// Mitsubishi GX Works2 project: NIAP1546_0600_IC-1M_R2   PLC: FX3S

PROGRAM MAIN
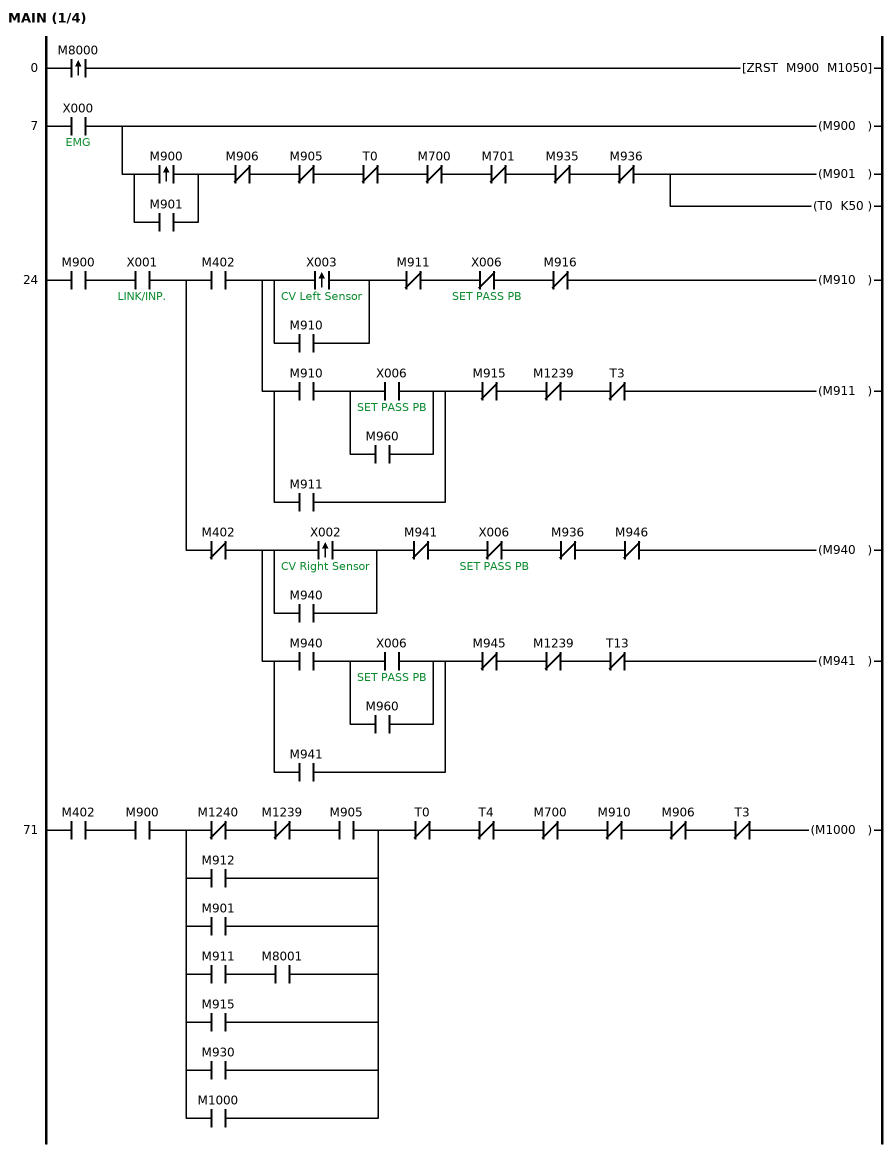
0     LDP     M8000
      ZRST    M900 M1050
7     LD      X000  ; EMG
      OUT     M900
      LDP     M900
      OR      M901
      ANB
      ANI     M906
      ANI     M905
      ANI     T0
      ANI     M700
      ANI     M701
      ANI     M935
      ANI     M936
      OUT     M901
      OUT     T0 K50
24    LD      M900
      AND     X001  ; LINK/INP.
      MPS
      AND     M402
      MPS
      LDP     X003  ; CV Left Sensor
      OR      M910
      ANB
      ANI     M911
      ANI     X006  ; SET PASS PB
      ANI     M916
      OUT     M910
      MPP
      LD      M910
      LD      X006  ; SET PASS PB
      OR      M960
      ANB
      OR      M911
      ANB
      ANI     M915
      ANI     M1239
      ANI     T3
      OUT     M911
      MPP
      ANI     M402
      MPS
      LDP     X002  ; CV Right Sensor
      OR      M940
      ANB
      ANI     M941
      ANI     X006  ; SET PASS PB
      ANI     M936
      ANI     M946
      OUT     M940
      MPP
      LD      M940
      LD      X006  ; SET PASS PB
      OR      M960
      ANB
      OR      M941
      ANB
      ANI     M945
      ANI     M1239
      ANI     T13
      OUT     M941
71    LD      M402
      AND     M900
      LDI     M1240
      ANI     M1239
      AND     M905
      OR      M912
      OR      M901
      LD      M911
      AND     M8001
      ORB
      OR      M915
      OR      M930
      OR      M1000
      ANB
      ANI     T0
      ANI     T4
      ANI     M700
      ANI     M910
      ANI     M906
      ANI     T3
      OUT     M1000
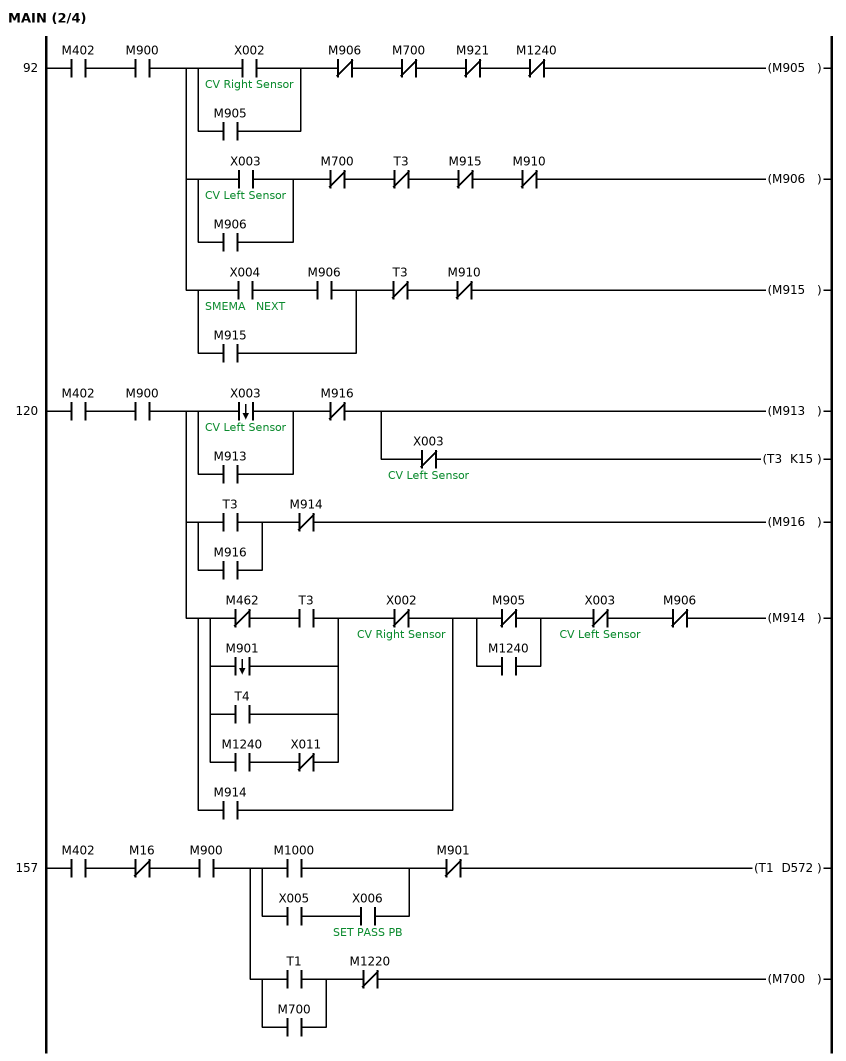
92    LD      M402
      AND     M900
      MPS
      LD      X002  ; CV Right Sensor
      OR      M905
      ANB
      ANI     M906
      ANI     M700
      ANI     M921
      ANI     M1240
      OUT     M905
      MRD
      LD      X003  ; CV Left Sensor
      OR      M906
      ANB
      ANI     M700
      ANI     T3
      ANI     M915
      ANI     M910
      OUT     M906
      MPP
      LD      X004  ; SMEMA   NEXT
      AND     M906
      OR      M915
      ANB
      ANI     T3
      ANI     M910
      OUT     M915
120   LD      M402
      AND     M900
      MPS
      LDF     X003  ; CV Left Sensor
      OR      M913
      ANB
      ANI     M916
      OUT     M913
      ANI     X003  ; CV Left Sensor
      OUT     T3 K15
      MRD
      LD      T3
      OR      M916
      ANB
      ANI     M914
      OUT     M916
      MPP
      LDI     M462
      AND     T3
      ORF     M901
      OR      T4
      LD      M1240
      ANI     X011
      ORB
      ANI     X002  ; CV Right Sensor
      OR      M914
      ANB
      LDI     M905
      OR      M1240
      ANB
      ANI     X003  ; CV Left Sensor
      ANI     M906
      OUT     M914
157   LD      M402
      ANI     M16
      AND     M900
      MPS
      LD      M1000
      LD      X005
      AND     X006  ; SET PASS PB
      ORB
      ANB
      ANI     M901
      OUT     T1 D572
      MPP
      LD      T1
      OR      M700
      ANB
      ANI     M1220
      OUT     M700
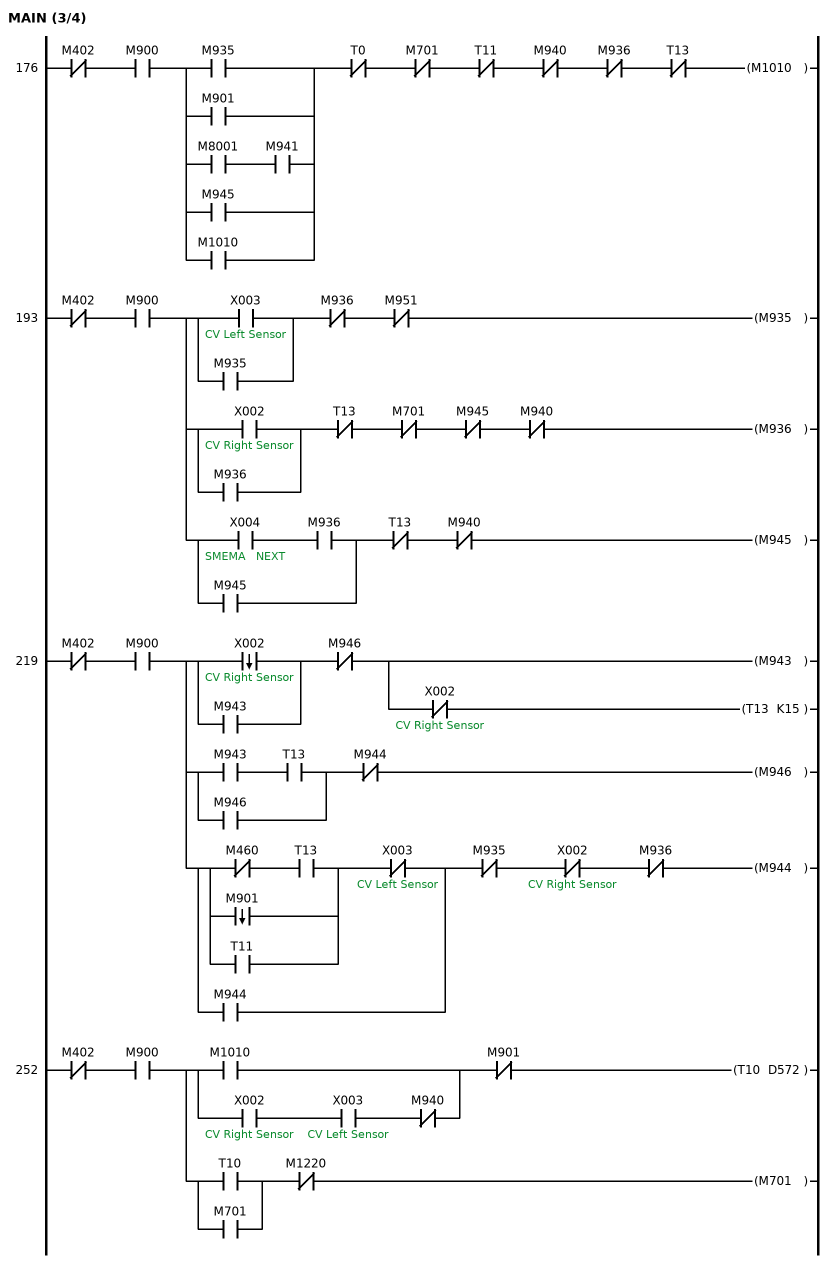
176   LDI     M402
      AND     M900
      LD      M935
      OR      M901
      LD      M8001
      AND     M941
      ORB
      OR      M945
      OR      M1010
      ANB
      ANI     T0
      ANI     M701
      ANI     T11
      ANI     M940
      ANI     M936
      ANI     T13
      OUT     M1010
193   LDI     M402
      AND     M900
      MPS
      LD      X003  ; CV Left Sensor
      OR      M935
      ANB
      ANI     M936
      ANI     M951
      OUT     M935
      MRD
      LD      X002  ; CV Right Sensor
      OR      M936
      ANB
      ANI     T13
      ANI     M701
      ANI     M945
      ANI     M940
      OUT     M936
      MPP
      LD      X004  ; SMEMA   NEXT
      AND     M936
      OR      M945
      ANB
      ANI     T13
      ANI     M940
      OUT     M945
219   LDI     M402
      AND     M900
      MPS
      LDF     X002  ; CV Right Sensor
      OR      M943
      ANB
      ANI     M946
      OUT     M943
      ANI     X002  ; CV Right Sensor
      OUT     T13 K15
      MRD
      LD      M943
      AND     T13
      OR      M946
      ANB
      ANI     M944
      OUT     M946
      MPP
      LDI     M460
      AND     T13
      ORF     M901
      OR      T11
      ANI     X003  ; CV Left Sensor
      OR      M944
      ANB
      ANI     M935
      ANI     X002  ; CV Right Sensor
      ANI     M936
      OUT     M944
252   LDI     M402
      AND     M900
      MPS
      LD      M1010
      LD      X002  ; CV Right Sensor
      AND     X003  ; CV Left Sensor
      ANI     M940
      ORB
      ANB
      ANI     M901
      OUT     T10 D572
      MPP
      LD      T10
      OR      M701
      ANB
      ANI     M1220
      OUT     M701
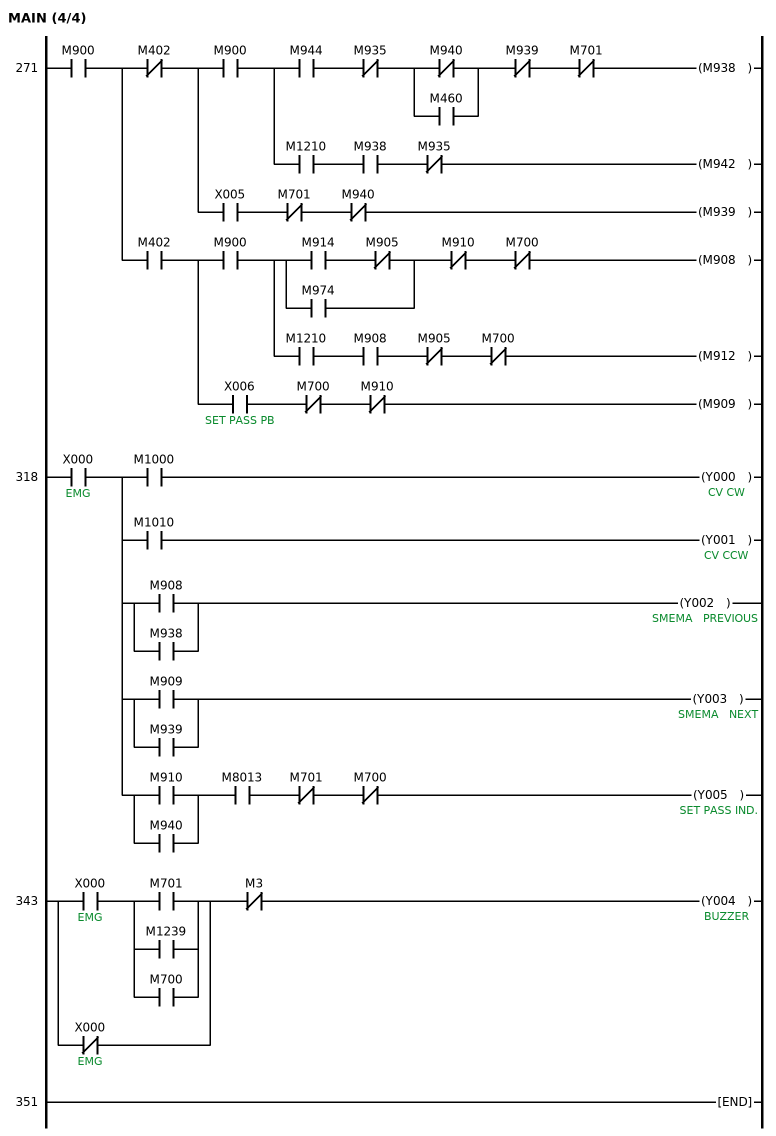
271   LD      M900
      MPS
      ANI     M402
      MPS
      AND     M900
      MPS
      AND     M944
      ANI     M935
      LDI     M940
      OR      M460
      ANB
      ANI     M939
      ANI     M701
      OUT     M938
      MPP
      AND     M1210
      AND     M938
      ANI     M935
      OUT     M942
      MPP
      AND     X005
      ANI     M701
      ANI     M940
      OUT     M939
      MPP
      AND     M402
      MPS
      AND     M900
      MPS
      LD      M914
      ANI     M905
      OR      M974
      ANB
      ANI     M910
      ANI     M700
      OUT     M908
      MPP
      AND     M1210
      AND     M908
      ANI     M905
      ANI     M700
      OUT     M912
      MPP
      AND     X006  ; SET PASS PB
      ANI     M700
      ANI     M910
      OUT     M909
318   LD      X000  ; EMG
      MPS
      AND     M1000
      OUT     Y000  ; CV CW
      MRD
      AND     M1010
      OUT     Y001  ; CV CCW
      MRD
      LD      M908
      OR      M938
      ANB
      OUT     Y002  ; SMEMA   PREVIOUS
      MRD
      LD      M909
      OR      M939
      ANB
      OUT     Y003  ; SMEMA   NEXT
      MPP
      LD      M910
      OR      M940
      ANB
      AND     M8013
      ANI     M701
      ANI     M700
      OUT     Y005  ; SET PASS IND.
343   LD      X000  ; EMG
      LD      M701
      OR      M1239
      OR      M700
      ANB
      ORI     X000  ; EMG
      ANI     M3
      OUT     Y004  ; BUZZER
351   END
END_PROGRAM
